// TwinCAT 3 PLC project Vibration_Test
// ProgramVersion: 3.1.4026.14
// CompilerDefines: VISU_USEPROPERTYINFO
// libraries:
//   Tc2_ControllerToolbox, * (Beckhoff Automation GmbH)
//   Tc2_Standard, * (Beckhoff Automation GmbH)
//   Tc2_System, * (Beckhoff Automation GmbH)
//   Tc2_Utilities, * (Beckhoff Automation GmbH)
// project tree:
//   / GlobalTextList.TcGTLO, PlcTask.TcTTO
//   POUs/ FB_PyListener.TcPOU, FB_UseScope.TcPOU, MAIN.TcPOU
//   VISUs/ Visualization.TcVIS, VisualizationManager.TcVMO (not stored)
// real-time tasks:
//   TASK PlcTask: cycle T#1ms, priority 20, ADS port 350
// I/O:
//   DEVICE Device 1 (EtherCAT), AmsNetId 192.168.1.5.2.1
//     Term 1 (EKM1101) [EKM1101 EtherCAT Coupler  (2A E-Bus, ID switch, Diagnostics, isolated)] (disabled)
//       Term 2 (ELM3604-0000) [ELM3604-0000 4Ch. IEPE Sensor, 24 bit, high precision]
//       Term 3 (EL9011) [EL9011 End Terminal]
//     AHU_RevE [m1sa]
// variable links:
//   Vibration_Test/Vibration_Test Instance <-> Device 1 (EtherCAT)/AHU_RevE
//     PlcTask Inputs/MAIN.saErrDongle <-> Status process data mapping/MAIN.saErrDongle
//     PlcTask Inputs/MAIN.saErrLocId <-> Status process data mapping/MAIN.saErrLocId
//     PlcTask Inputs/MAIN.saErrMasterHb <-> Status process data mapping/MAIN.saErrMasterHb
//     PlcTask Inputs/MAIN.saForceSpX <-> Status process data mapping/MAIN.saForceSpX
//     PlcTask Inputs/MAIN.saPwm1 <-> Status process data mapping/MAIN.saPwm1
//     PlcTask Outputs/MAIN.saClearFault <-> Control process data mapping/MAIN.saClearFault
//     PlcTask Outputs/MAIN.saCloseLoop <-> Control process data mapping/MAIN.saCloseLoop
//     PlcTask Outputs/MAIN.saEnable <-> Control process data mapping/MAIN.saEnable
//     PlcTask Outputs/MAIN.saForceSetting <-> Control process data mapping/MAIN.saForceSetting
//     PlcTask Outputs/MAIN.saMsthb <-> Control process data mapping/MAIN.saMsthb
//   Vibration_Test/Vibration_Test Instance <-> Device 1 (EtherCAT)/Term 1 (EKM1101)/Term 2 (ELM3604-0000)
//     PlcTask Inputs/MAIN.ZAxisNumSamples <-> PAI Status Channel 3/Status/MAIN.ZAxisNumSamples
//     PlcTask Inputs/MAIN.errXAxisOverRnge <-> PAI Status Channel 1/Status/MAIN.errXAxisOverRnge
//     PlcTask Inputs/MAIN.errXAxisSample <-> PAI Status Channel 1/Status/MAIN.errXAxisSample
//     PlcTask Inputs/MAIN.errXAxisUndrRnge <-> PAI Status Channel 1/Status/MAIN.errXAxisUndrRnge
//     PlcTask Inputs/MAIN.errYAxisOverRnge <-> PAI Status Channel 2/Status/MAIN.errYAxisOverRnge
//     PlcTask Inputs/MAIN.errYAxisSample <-> PAI Status Channel 2/Status/MAIN.errYAxisSample
//     PlcTask Inputs/MAIN.errYAxisUndrRnge <-> PAI Status Channel 2/Status/MAIN.errYAxisUndrRnge
//     PlcTask Inputs/MAIN.errZAxisOverRnge <-> PAI Status Channel 3/Status/MAIN.errZAxisOverRnge
//     PlcTask Inputs/MAIN.errZAxisSample <-> PAI Status Channel 3/Status/MAIN.errZAxisSample
//     PlcTask Inputs/MAIN.errZAxisUndrRnge <-> PAI Status Channel 3/Status/MAIN.errZAxisUndrRnge
//     PlcTask Inputs/MAIN.xAxisNumSamples <-> PAI Status Channel 1/Status/MAIN.xAxisNumSamples
//     PlcTask Inputs/MAIN.xAxisReadingRaw <-> PAI Samples 1 Channel 1/Samples[0]
//     PlcTask Inputs/MAIN.yAxisNumSamples <-> PAI Status Channel 2/Status/MAIN.yAxisNumSamples
//     PlcTask Inputs/MAIN.yAxisReadingRaw <-> PAI Samples 1 Channel 2/Samples[0]
//     PlcTask Inputs/MAIN.zAxisReadingRaw <-> PAI Samples 1 Channel 3/Samples[0]

CONFIGURATION Vibration_Test
    RESOURCE PLC ON TwinCAT3
        TASK PlcTask(INTERVAL := T#1ms, PRIORITY := 20);
        PROGRAM MAIN WITH PlcTask : MAIN;
    END_RESOURCE
END_CONFIGURATION

// ---- POUs/MAIN.TcPOU
PROGRAM MAIN
VAR
	bInit								: BOOL := TRUE;
	
	tSigGenTimer						: TON;
	tTestTimer							: TON;
	
	fbPyListen							: FB_PyListener;
	pyLoadBusy							: BOOL := FALSE;
	pyReady								: BOOL := FALSE;
	tglPyTest							: BOOL;
	sPyTestMsg 							: STRING := 'Run Data Collection';
	
	fbSigGen							: FB_CTRL_SIGNAL_GENERATOR;
	stCTRL_SIGNAL_GENERATOR_PARAMS		: ST_CTRL_SIGNAL_GENERATOR_PARAMS;
	sigType								: E_CTRL_SIGNAL_TYPE;
	eMode								: E_CTRL_MODE;
	bUseSigGen							: BOOL := FALSE;
	sigGenFreq							: REAL := 10;
	sigGenTime							: REAL;
	
	fbUseScope							: FB_UseScope;
	fbScopeServerControl				: FB_ScopeServerControl;
    eReqState							: E_ScopeServerState := SCOPE_SERVER_IDLE;
	bBusy								: BOOL := FALSE;
    bDone								: BOOL := FALSE;
    bError								: BOOL := FALSE;
    nErrorId							: UDINT := 0;
	
	// Support actuator board control variables
	saMsthb	AT %Q*						: UDINT := 0;
	saEnable AT %Q*						: BOOL := FALSE;
	saCloseLoop AT %Q*					: BOOL := TRUE;
	saClearFault AT %Q*					: BOOL := FALSE;
	saForceSetting AT %Q*				: REAL := 0;
	
	// Support actuator board monitor variables
	saForceSpX AT %I*					: REAL := 0;
	saPwm1 AT %I*						: INT;
	saErrMasterHb AT %I*				: BOOL;
	saErrDongle	AT %I*					: BOOL;
	saErrLocId AT %I*					: BOOL;		

	// Accelerometer measurement and status variables
	xAxisReadingRaw AT %I* 				: DINT; // Raw measurement from acccelerometers are in nV
	yAxisReadingRaw AT %I* 				: DINT;
	zAxisReadingRaw AT %I*				: DINT;
	
	xAxisConverted_g					: REAL; // Converted accelerometer readings to g
	yAxisConverted_g					: REAL;
	zAxisConverted_g					: REAL;
	
	xAxisConverted_mps2					: REAL; // Converted accelerometer readings to m/s
	yAxisConverted_mps2					: REAL;
	zAxisConverted_mps2					: REAL;
	
	// Accelerometer status variables
	xAxisNumSamples AT %I*				: USINT;
	errXAxisSample AT %I*				: BOOL;
	errXAxisOverRnge AT %I*				: BOOL;
	errXAxisUndrRnge AT %I*				: BOOL;
	
	yAxisNumSamples AT %I*				: USINT;
	errYAxisSample AT %I*				: BOOL;
	errYAxisOverRnge AT %I*				: BOOL;
	errYAxisUndrRnge AT %I*				: BOOL;
	
	ZAxisNumSamples AT %I*				: USINT;
	errZAxisSample AT %I*				: BOOL;
	errZAxisOverRnge AT %I*				: BOOL;
	errZAxisUndrRnge AT %I*				: BOOL;
	
	test								: BOOL;

END_VAR

VAR CONSTANT	
	Accelerometer_Coefficient_16 		: REAL := ((9.8 / 2) / 65536); 		//Max INT is 2^16, and the accelerometers can only do 0.5g fullscale
	Accelerometer_Coefficient_24 		: REAL := ((9.8 / 2) / 16777213); 	//Max INT is 2^24, and the accelerometers can only do 0.5g fullscale
END_VAR

saMsthb := saMsthb + 1; // Support actuator heartbeat increment

//fbUseScope(bExternalTriggerEvent := test);
(*
fbScopeServerControl( sNetId:= '',
                      eReqState:= eReqState,
                      //sConfigFile:= 'C:\twinCat\scope\test.sv2',
                      //sSaveFile:= 'C:\twinCat\scope\test.svd',
                      tTimeout:= t#5s,
                      bBusy=>bBusy,
                      bDone=>bDone,
                      bError=>bError,
                      nErrorId=>nErrorId);
*)

// Initialization routine, run once, set up signal generator setpoints
IF bInit THEN
	(* init the setpoint array *)
	stCTRL_SIGNAL_GENERATOR_PARAMS.tCtrlCycleTime := T#1MS;
	stCTRL_SIGNAL_GENERATOR_PARAMS.tTaskCycleTime := T#1MS;
	stCTRL_SIGNAL_GENERATOR_PARAMS.eSignalType := 1; // Sine wave
	stCTRL_SIGNAL_GENERATOR_PARAMS.tStart := T#0S;
	stCTRL_SIGNAL_GENERATOR_PARAMS.tCylceDuration := T#1S; // Default period of 1s or 10Hz
	stCTRL_SIGNAL_GENERATOR_PARAMS.fAmplitude := 80; // Amplitude of sinewave
	stCTRL_SIGNAL_GENERATOR_PARAMS.fOffset := 0;

	(* reset init flag *)
	bInit := FALSE;
END_IF

IF tglPyTest = TRUE THEN

	//fbPyListen(bExecute := TRUE); // Launch Python data collection code when button is pressed
	//pyLoadBusy := TRUE; // Flag for if Python collection is busy collecting data, watched in Py script
	pyReady := TRUE;
	IF pyReady = TRUE THEN
		
		//fbUseScope(bExternalTriggerEvent := pyReady);
		tSigGenTimer(IN := TRUE, PT := T#1mS);
		tTestTimer(IN := TRUE, PT := T#120S);

		IF tSigGenTimer.Q = TRUE THEN
			bUseSigGen := TRUE;
		END_IF
	
		IF tTestTimer.Q = TRUE THEN
		(*	fbPyListen(
				Initialized := FALSE,
				bExecute := FALSE,
				Init_State := 0
				); *)
			tTestTimer(IN := FALSE);
			tSigGenTimer(IN := FALSE);
			//PyLoadBusy := FALSE;
			bUseSigGen := FALSE;
			tglPyTest := FALSE;
			saForceSetting := 0;
			pyReady := FALSE;
		END_IF
	
	END_IF
END_IF

IF saEnable = TRUE AND bUseSigGen = TRUE THEN
	// Convert from Hz to time, scale to get appropriate ms
	//stCTRL_SIGNAL_GENERATOR_PARAMS.tCylceDuration := REAL_TO_TIME((1 / sigGenFreq) * 10000);
	sigGenTime := 1 / sigGenFreq;
	stCTRL_SIGNAL_GENERATOR_PARAMS.tCylceDuration := REAL_TO_TIME(sigGenTime * 1000);
	// Signal generator function to generate sine wave using defined properties, send to force setpoint
	fbSigGen(
		stParams := stCTRL_SIGNAL_GENERATOR_PARAMS,
		eMode := eCTRL_MODE_ACTIVE, // Set the mode to ACTIVE --> normal operation
		fOut => saForceSetting,
	);	
ELSIF saEnable = FALSE AND bUseSigGen = TRUE THEN
	// Reset signal generator back to 0 for next card enable with signal generator
	fbSigGen(
		stParams := stCTRL_SIGNAL_GENERATOR_PARAMS,
		eMode := eCTRL_MODE_RESET);
END_IF

saPwm1 := saPwm1 / 100; // Convert PWM signal to percent

(*
xAxisConvertedG := 0.1 * (DINT_TO_REAL(xAxisReadingRaw) * 10E-9); // (g/10V) * (nV * 10^-9 V/nV)
yAxisConvertedG := 0.1 * (DINT_TO_REAL(yAxisReadingRaw) * 10E-9);
zAxisConvertedG := 0.1 * (DINT_TO_REAL(zAxisReadingRaw) * 10E-9);
*)
(*
// Convert accelerometer data to m/s^2
xAxisConverted_mps2 := DINT_TO_REAL(xAxisReadingRaw) * Accelerometer_Coefficient_16; 
yAxisConverted_mps2 := DINT_TO_REAL(yAxisReadingRaw) * Accelerometer_Coefficient_16;
zAxisConverted_mps2 := DINT_TO_REAL(zAxisReadingRaw) * Accelerometer_Coefficient_16;

// Convert accelerometer from m/s^2 to g
xAxisConverted_g := DINT_TO_REAL(xAxisReadingRaw) * Accelerometer_Coefficient_16 * 0.10197162;
yAxisConverted_g := DINT_TO_REAL(yAxisReadingRaw) * Accelerometer_Coefficient_16 * 0.10197162;
zAxisConverted_g := DINT_TO_REAL(zAxisReadingRaw) * Accelerometer_Coefficient_16 * 0.10197162;
*)

xAxisConverted_g := (DINT_TO_REAL(xAxisReadingRaw) / 7812500) / 9.65;
yAxisConverted_g := (DINT_TO_REAL(yAxisReadingRaw) / 7812500) / 9.8;
zAxisConverted_g := (DINT_TO_REAL(zAxisReadingRaw) / 7812500) / 10; // Sensitivity inknown, cal card not with accelerometer

xAxisConverted_mps2 := (DINT_TO_REAL(xAxisReadingRaw) / 7812500) / 1.02;
yAxisConverted_mps2 := (DINT_TO_REAL(yAxisReadingRaw) / 7812500) / 1.02;
zAxisConverted_mps2 := (DINT_TO_REAL(zAxisReadingRaw) / 7812500) / 1.02;

END_PROGRAM

// ---- POUs/FB_PyListener.TcPOU
FUNCTION_BLOCK FB_PyListener
VAR_INPUT
	bExecute			: BOOL := FALSE;
	Initialized 		: BOOL := FALSE;
	Init_State  		: UINT := 0;
END_VAR
VAR_OUTPUT
	bIsBusy				: BOOL;
    ERR             	: BOOL;
    ERRID           	: UDINT;
END_VAR
VAR
	Process         	: NT_StartProcess;
	RisingEdge			: R_TRIG;
	bError          	: BOOL;
    sTargetFilePath     : STRING(255);
    sTargetDirectory    : STRING(255);
    sCommand        	: STRING(255);
    iErrorId            : UDINT; 	
END_VAR

IF NOT Initialized THEN
  (* Initialization State Machine *)
  CASE Init_State OF
    0: (* First step in initialization *)
	
		// File Locations
		sTargetDirectory := 'C:\Vibration_Testing\Actuator_Testing\Scripts\';
 
		// Build Command String                 
		// Special command indicating command string input
		sCommand := CONCAT(sTargetDirectory, 'TwinCAT_DataCollector.py');      // Execute Python data collection script
        Init_State := Init_State + 1;
	   
    1: (* Second step in initialization *)
		Process(
    	NETID := '',                    					// Local System
		//PATHSTR := 'C:\ProgramData\Anaconda3\python.exe',   // Path to local cmd executable
		PATHSTR := 'py',
		//PATHSTR := 'python',
    	COMNDLINE := sCommand,          					// Comnmand to be executed
    	ERR => bError,                   					// Error Output
    	ERRID => iErrorId,                					// Error Id Output
		BUSY => bIsBusy,									// Process is already busy, used to not call multiple instances
		START := TRUE
		);
        Init_State := Init_State + 1;

    2: (* Last step in initialization *)
		Process(START := FALSE);
		bExecute := FALSE;
		RisingEdge.CLK := FALSE;
        Initialized := TRUE;
  END_CASE
END_IF

END_FUNCTION_BLOCK

// ---- POUs/FB_UseScope.TcPOU
FUNCTION_BLOCK FB_UseScope
VAR_INPUT
    bExternalTriggerEvent			: BOOL := FALSE;
	nState							: UDINT := 0;
END_VAR
VAR_OUTPUT
END_VAR
VAR
    fbScopeServerControl			: FB_ScopeServerControl;
    eReqState						: E_ScopeServerState := SCOPE_SERVER_IDLE;
    bBusy							: BOOL := FALSE;
    bDone							: BOOL := FALSE;
    bError							: BOOL := FALSE;
    nErrorId						: UDINT := 0;
    fbTimer							: TON;
    bTriggerTimer					: BOOL := FALSE;
END_VAR

(*
CASE nState OF
0:
    eReqState := SCOPE_SERVER_START;
    nState := nState + 1;
1:
    IF fbScopeServerControl.bDone AND bExternalTriggerEvent
    THEN
        bTriggerTimer := TRUE;
		nState := nState + 1;
    END_IF
2:
    IF fbTimer.Q THEN
        eReqState := SCOPE_SERVER_SAVE;
        bTriggerTimer := FALSE;
        nState := nState + 1;
    END_IF
3:
    IF fbScopeServerControl.bDone THEN
        eReqState := SCOPE_SERVER_DISCONNECT;
    END_IF
END_CASE

fbTimer(IN:=bTriggerTimer, PT:=T#10S);
*)
fbScopeServerControl( sNetId:= '192.168.1.14.1.1',
                      eReqState:= eReqState,
                      //sConfigFile:= 'C:\twinCat\scope\test.sv2',
                      //sSaveFile:= 'C:\twinCat\scope\test.svd',
                      tTimeout:= t#5s,
                      bBusy=>bBusy,
                      bDone=>bDone,
                      bError=>bError,
                      nErrorId=>nErrorId);

END_FUNCTION_BLOCK

// ---- GlobalTextList.TcGTLO
TEXTLIST GlobalTextList
  838 = '%5.3f'
  947 = '%s'
  978 = 'Clear SA Faults'
  99 = 'Collect Data'
  747 = 'Desired SA Force'
  130 = 'Dongle Error'
  385 = 'Enable SA Card'
  104 = 'Err Num Samples'
  62 = 'Err Over Range'
  1 = 'Err Sample'
  685 = 'Err Under Range'
  897 = 'Err X Axis Num Samples'
  344 = 'Err X Axis Sample'
  614 = 'Err X Axis Samples'
  70 = 'Location ID Error'
  287 = 'Master Heartbeat Error'
  95 = 'Num. Samples'
  549 = 'PWM Output'
  197 = 'SA Force'
  14 = 'Signal Generator Amplitude'
  988 = 'Signal Generator Freq [Hz]'
  165 = 'Use Signal Generator'
  407 = 'X-Axis'
  762 = "X-Axis (G's)"
  155 = 'X-Axis [g]'
  806 = 'X-Axis [m/s^2]'
  2 = 'Y-Axis'
  138 = 'Y-Axis  [g]'
  453 = "Y-Axis (G's)"
  332 = 'Y-Axis [m/s^2]'
  773 = 'Z-Axis'
  910 = 'Z-Axis  [g]'
  318 = "Z-Axis (G's)"
  312 = 'Z-Axis [m/s^2]'
END_TEXTLIST

// ---- VISUs/Visualization.TcVIS
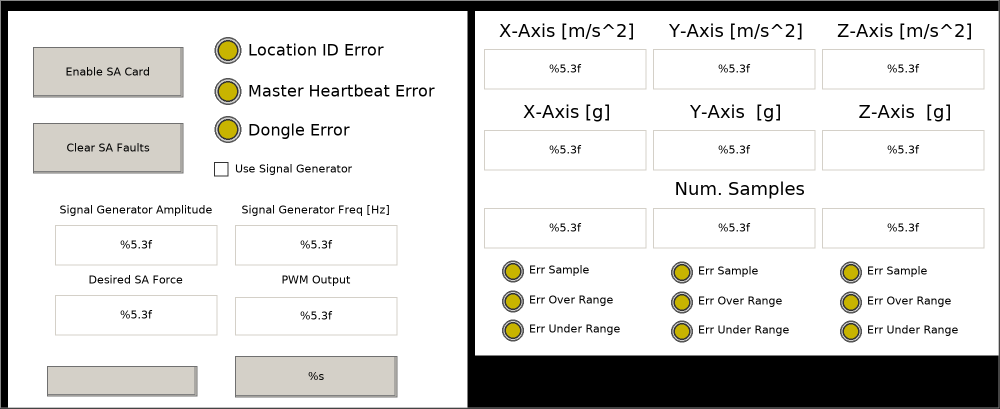
VISUALIZATION Visualization  // 1000x409
    RoundedRectangle (7,10 461x399)
    RoundedRectangle (474,10 526x346)
    Lamp1 (212,76 32x31), variable: MAIN.saErrMasterHb, style: Lamp-Lamp1-Yellow
    Lamp1 (212,114 32x31), variable: MAIN.saErrDongle, style: Lamp-Lamp1-Yellow
    Label (245,76 213x30), "Master Heartbeat Error"
    Label (245,115 213x30), "Dongle Error"
    Button (33,47 150x50), "Enable SA Card"
        toggle MAIN.saEnable
    Textfield (55,295 162x40), "%5.3f", text variable: MAIN.saForceSetting
        OnMouseClick: write MAIN.saForceSetting via Default
    Label (61,265 150x30), "Desired SA Force"
    Button (33,123 150x50), "Clear SA Faults"
        tap MAIN.saClearFault
    Textfield (235,297 162x38), "%5.3f", text variable: MAIN.saPwm1
    Label (241,265 150x30), "PWM Output"
    Label (492,97 150x30), "X-Axis [g]"
    Textfield (484,130 162x40), "%5.3f", text variable: MAIN.xAxisConverted_g
    Label (661,97 150x30), "Y-Axis [g]"
    Textfield (653,130 162x40), "%5.3f", text variable: MAIN.yAxisConverted_g
    Label (830,97 150x30), "Z-Axis [g]"
    Textfield (822,130 162x40), "%5.3f", text variable: MAIN.zAxisConverted_g
    Label (665,174 150x30), "Num. Samples"
    Textfield (484,208 162x40), "%5.3f", text variable: MAIN.xAxisNumSamples
    Textfield (653,208 162x40), "%5.3f", text variable: MAIN.yAxisNumSamples
    Textfield (822,208 162x40), "%5.3f", text variable: MAIN.ZAxisNumSamples
    Label (526,255 124x30), "Err Sample"
    Lamp1 (496,259 34x25), variable: MAIN.errXAxisSample, style: Lamp-Lamp1-Yellow
    Label (526,285 124x30), "Err Over Range"
    Lamp1 (496,289 34x25), variable: MAIN.errXAxisOverRnge, style: Lamp-Lamp1-Yellow
    Label (526,314 124x30), "Err Under Range"
    Lamp1 (496,318 34x25), variable: MAIN.errXAxisUndrRnge, style: Lamp-Lamp1-Yellow
    Label (695,256 124x30), "Err Sample"
    Lamp1 (665,260 34x25), variable: MAIN.errYAxisSample, style: Lamp-Lamp1-Yellow
    Label (695,286 124x30), "Err Over Range"
    Lamp1 (665,290 34x25), variable: MAIN.errYAxisOverRnge, style: Lamp-Lamp1-Yellow
    Label (695,315 124x30), "Err Under Range"
    Lamp1 (665,319 34x25), variable: MAIN.errYAxisUndrRnge, style: Lamp-Lamp1-Yellow
    Label (864,256 124x30), "Err Sample"
    Lamp1 (834,260 34x25), variable: MAIN.errZAxisSample, style: Lamp-Lamp1-Yellow
    Label (864,286 124x30), "Err Over Range"
    Lamp1 (834,290 34x25), variable: MAIN.errZAxisOverRnge, style: Lamp-Lamp1-Yellow
    Label (864,315 124x30), "Err Under Range"
    Lamp1 (834,319 34x25), variable: MAIN.errYAxisUndrRnge, style: Lamp-Lamp1-Yellow
    Button (235,356 162x41), "%s", text variable: MAIN.sPyTestMsg
        toggle MAIN.tglPyTest
    Lamp1 (212,35 32x31), variable: MAIN.saErrLocId, style: Lamp-Lamp1-Yellow
    Label (245,35 213x30), "Location ID Error"
    Checkbox (212,154 234x30), "Use Signal Generator", variable: MAIN.bUseSigGen
    Label (241,195 150x30), "Signal Generator Freq [Hz]"
    Textfield (235,225 162x40), "%5.3f", text variable: MAIN.sigGenFreq
        OnMouseClick: write MAIN.sigGenFreq via Default
    Label (492,16 150x30), "X-Axis [m/s^2]"
    Textfield (484,49 162x40), "%5.3f", text variable: MAIN.xAxisConverted_mps2
    Label (661,16 150x30), "Y-Axis [m/s^2]"
    Textfield (653,49 162x40), "%5.3f", text variable: MAIN.yAxisConverted_mps2
    Label (830,16 150x30), "Z-Axis [m/s^2]"
    Textfield (822,49 162x40), "%5.3f", text variable: MAIN.zAxisConverted_mps2
    Label (61,195 150x30), "Signal Generator Amplitude"
    Textfield (55,225 162x40), "%5.3f", text variable: MAIN.stCTRL_SIGNAL_GENERATOR_PARAMS.fAmplitude
        OnMouseClick: write MAIN.stCTRL_SIGNAL_GENERATOR_PARAMS.fAmplitude via Default
    Button (47,366 150x30)
        toggle MAIN.test
END_VISUALIZATION
